// TIA Portal V20 export
FUNCTION_BLOCK "FB_IO_Device_Functional_Test_Rework"   // FB12, LAD
{ S7_Optimized_Access := 'TRUE' }
// stored: AutoNumber false, MemoryReserve 100, SetENOAutomatically false
   VAR_INPUT
      Reset_PLC_Functional_Test_Rework : Bool;
      Status : Bool;
      Voltage_Read : UInt;
      Min_Electrical_Current : UInt;
      Max_Electrical_Current : UInt;
      Time_End_Electrical_Current_Test : Time;
      Time_Start_Visual_Test : Time;
      In_Functional_Test_Rework : "IO_Device_Functinal_Test_Rework";
   END_VAR
   VAR_OUTPUT
      Out_Test_Parameters_Rework : "IO_Device_Test_Parameters_Rework";
      Comunication_Error_Panel_Rework : Bool;
   END_VAR
   VAR
      Timer_Alarme_A_1 { S7_SetPoint := 'True'} : TON_TIME;
      Timer_Alarme_B_1 { S7_SetPoint := 'True'} : TON_TIME;
   END_VAR
BEGIN

REGION Network 1
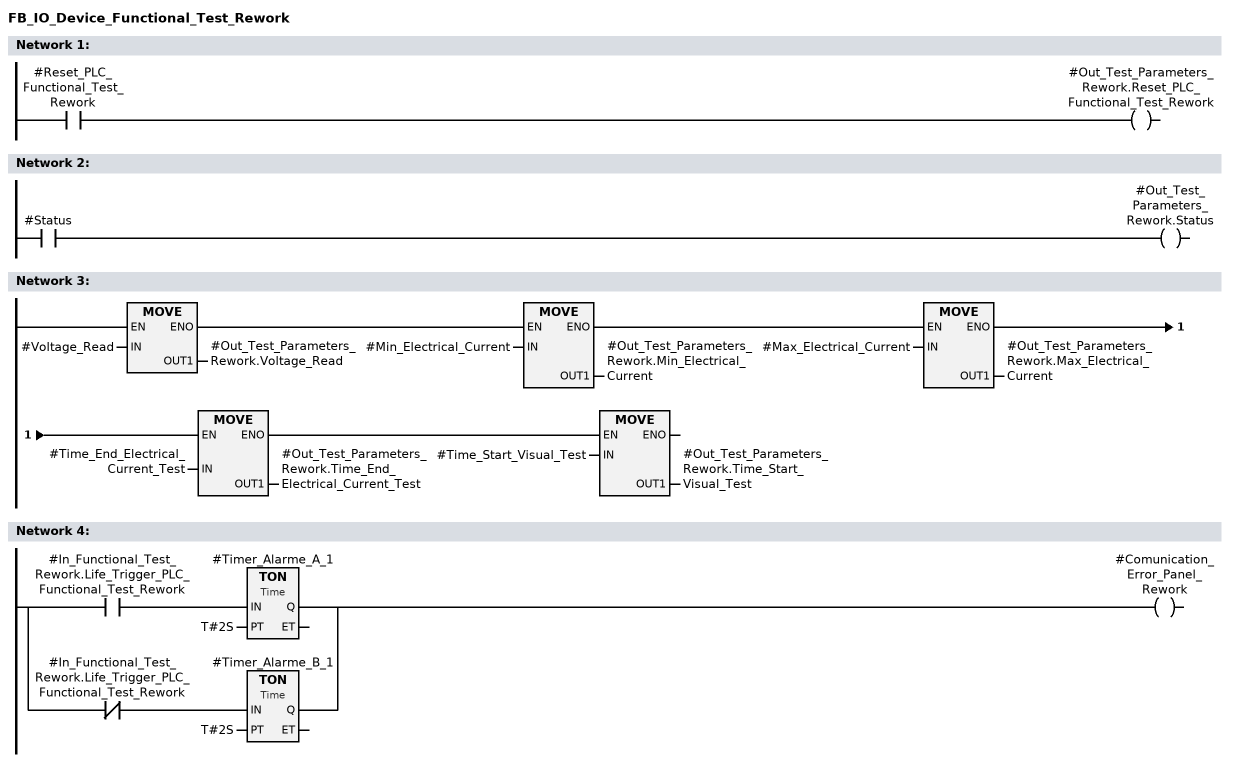
   RUNG wire#powerrail
      Contact( #Reset_PLC_Functional_Test_Rework )
      Coil( #Out_Test_Parameters_Rework.Reset_PLC_Functional_Test_Rework )
   END_RUNG
   // the same network as SCL:
   #Out_Test_Parameters_Rework.Reset_PLC_Functional_Test_Rework := #Reset_PLC_Functional_Test_Rework;
END_REGION

REGION Network 2
   RUNG wire#powerrail
      Contact( #Status )
      Coil( #Out_Test_Parameters_Rework.Status )
   END_RUNG
   // the same network as SCL:
   #Out_Test_Parameters_Rework.Status := #Status;
END_REGION

REGION Network 3
   RUNG wire#powerrail
      Move(in := #Voltage_Read, out1 => #Out_Test_Parameters_Rework.Voltage_Read)
      Move(in := #Min_Electrical_Current, out1 => #Out_Test_Parameters_Rework.Min_Electrical_Current)
      Move(in := #Max_Electrical_Current, out1 => #Out_Test_Parameters_Rework.Max_Electrical_Current)
      Move(in := #Time_End_Electrical_Current_Test, out1 => #Out_Test_Parameters_Rework.Time_End_Electrical_Current_Test)
      Move(in := #Time_Start_Visual_Test, out1 => #Out_Test_Parameters_Rework.Time_Start_Visual_Test)
   END_RUNG
   // the same network as SCL:
   #Out_Test_Parameters_Rework.Voltage_Read := #Voltage_Read;
   #Out_Test_Parameters_Rework.Min_Electrical_Current := #Min_Electrical_Current;
   #Out_Test_Parameters_Rework.Max_Electrical_Current := #Max_Electrical_Current;
   #Out_Test_Parameters_Rework.Time_End_Electrical_Current_Test := #Time_End_Electrical_Current_Test;
   #Out_Test_Parameters_Rework.Time_Start_Visual_Test := #Time_Start_Visual_Test;
END_REGION

REGION Network 4
   RUNG wire#powerrail
      Contact( #In_Functional_Test_Rework.Life_Trigger_PLC_Functional_Test_Rework )
      { S7_Templates := "time_type := Time" } #Timer_Alarme_A_1.TON(pt := T#2S, et =>)
      wire#w1
      Coil( #Comunication_Error_Panel_Rework )
   END_RUNG
   RUNG wire#powerrail
      I_Contact( #In_Functional_Test_Rework.Life_Trigger_PLC_Functional_Test_Rework )
      { S7_Templates := "time_type := Time" } #Timer_Alarme_B_1.TON(pt := T#2S, et =>)
   END_RUNG wire#w1
   // the same network as SCL:
   #Timer_Alarme_A_1(IN := #In_Functional_Test_Rework.Life_Trigger_PLC_Functional_Test_Rework, PT := T#2S);   // TON
   #Timer_Alarme_B_1(IN := NOT #In_Functional_Test_Rework.Life_Trigger_PLC_Functional_Test_Rework, PT := T#2S);   // TON
   #Comunication_Error_Panel_Rework := #Timer_Alarme_A_1.Q OR #Timer_Alarme_B_1.Q;
END_REGION
END_FUNCTION_BLOCK
